PROGRAM P_Demo_F_ARGISZERO
VAR
    nLiveValue     : INT := 42; // 业务值
    argInUse       : T_Arg; // 会被 F_INT 绑定的槽位
    argUnused      : T_Arg; // 不绑定，模拟空槽位
    bInUseIsEmpty  : BOOL; // 期望 FALSE
    bUnusedIsEmpty : BOOL; // 期望 TRUE
    bCheck         : BOOL; // 在线置 TRUE 触发一次检查
END_VAR

// ============================================================
// Tc2_Utilities.F_ARGISZERO 演示程序
// ============================================================
// 场景：遍历 T_ArgList 时跳过未填的空槽位，避免 deref pData=0 崩溃。
// 价值：一行替代 IF a.pData = 0 OR a.cbLen = 0 OR a.eType = 0 THEN 三段判空。
// 验证：bCheck := TRUE；bInUseIsEmpty 应为 FALSE，bUnusedIsEmpty 应为 TRUE。
// ============================================================

// 只绑定 argInUse；argUnused 保持默认（三字段都为 0）
argInUse := F_INT(nLiveValue);

IF bCheck THEN
    bInUseIsEmpty  := F_ARGISZERO(arg := argInUse);
    bUnusedIsEmpty := F_ARGISZERO(arg := argUnused);
    bCheck := FALSE;
END_IF;

END_PROGRAM

(* stored: Version 1.1.0.1, ProductVersion 3.1.4024.5
   POU P_Demo_F_ARGISZERO: Id {15d044a3-8f0e-53fb-86c6-73f89d390bab}, SpecialFunc None *)
